// TIA Portal V17 export
// export: Created 2024-09-02T12:50:31.7482336Z, ExportSetting WithDefaults, DisplayName Totally Integrated Automation Portal, DisplayVersion V17, DisplayName TIA Portal Openness, DisplayVersion V17, DisplayName TIA Portal Version Control Interface, DisplayVersion V17, DisplayName STEP 7 Professional, DisplayVersion V17, DisplayName STEP 7 Safety, DisplayVersion V17, DisplayName WinCC Professional, DisplayVersion V17
TYPE "UFM_StationStatus"
TITLE = UFM_StationStatus
// Describes the current status of the UFM station.
// stored: IsFailsafeCompliant false
   STRUCT
      SignalLimitTooEarly : Bool;
      SignalLimitNotReached : Bool;
      MeasuredValueNotCaptured : Bool;
      MeasuredValueUpperLimitViolated : Bool;
      MeasuredValueLowerLimitViolated : Bool;
      FollowingError : Bool;
      MaximumPosition : Bool;
      UpperEnvelopeCurveViolated : Bool;
      LowerEnvelopeCurveViolated : Bool;
      CurveMemoryOverrun : Bool;
      TriggerFunctionError : Bool;
      NcModuleError : Bool;
      NcSetOkManually : Bool;
      NcSetNokManually : Bool;
      SensorOffsetError : Bool;
      Overload : Bool;
      HomingError : Bool;
      EmergencyOff : Bool;
      StartSignalLost : Bool;
      NoProgramLoaded : Bool;
      MaxPositionReached : Bool;
      NcModuleReset : Bool;
      ConverterTrip : Bool;
      AdcOverload : Bool;
      CtNetCouplerError : Bool;
      MotorOverload : Bool;
      SConfig : Bool;
      SignalSource_1_Value : Real;
      SignalSource_2_Value : Real;
      SignalSource_3_Value : Real;
      UserOutput : Word;
      CurrentProgram : Word;
      ReferenceRequest : Bool;
      ReadyToStart : Bool;
      CurveDataReady : Bool;   // Curve data ready to be retrieved (by UDP library)
      PiezoOperational : Bool;   // OP_PIEZO status bit of the station. Indicates if the piezo preamplifier is in its operational state.
      PiezoOperationalState : Bool;   // Current state of the piezo output of the library, i.e. the value last set with UFM_SetPiezoState.
      PcLive : Bool;   // Gibt an, ob der PC mit UFM Software mit dem Applikationsmodul verbunden ist oder nicht.
      MeasuredValueLeftLimitViolated : Bool;
      MeasuredValueRightLimitViolated : Bool;
      Straincompensation : Bool;
      Brake : Bool;
      AxisLocked : Bool;
   END_STRUCT;
END_TYPE
